// TIA Portal V21 export
VAR_GLOBAL   // PLC tag table "K_RicettaSterilizzatoreTubo"
END_VAR
VAR_GLOBAL CONSTANT   // user constants
   K_DatoRicettaBool_SterilizzatoreTubo_AbilitazionePompaPistoni : Int := 1;
   K_NumDatoRicettaBool_SterilizzatoreTubo : Int := 1;
   K_NumDatoRicettaReal_SterilizzatoreTubo : Int := 3;
   K_DatoRicettaReal_SterilizzatoreTubo_m³TubazioneRiempi : Int := 1;
   K_DatoRicettaReal_SterilizzatoreTubo_m³TubazioneSvuota : Int := 2;
   K_DatoRicettaReal_SterilizzatoreTubo_ContropressioneFiltri : Int := 3;
END_VAR
